// TIA Portal V18 export
TYPE "UDT_vDI"
// stored: IsFailsafeCompliant false
   STRUCT
      xInput : Bool;
      xMemoryIn : Bool;   // Temp
      xMemoryOut : Bool;
      xInversion : Bool;   // DIs label for monitoring
      xOutput : Bool;   // Filtered value
      xtemp1 : Bool;
      xtemp2 : Bool;
      xtemp3 : Bool;
      cMemory : Byte := 0;
      iCounterOut : Int;
      iCounterIn : Int;   // Counter for DIs EDGE
      cFuncSystemID : Byte := 0;
      cFuncVar : Byte := 0;
      cDelayOnSec : Byte := 0;   // Temp
      cDelayOffSec : Byte := 0;   // Temp
   END_STRUCT;
END_TYPE
